// TIA Portal project "RUNNING_ A_PUMP" (V16)

(* hardware
DEVICE "S7-1200 station_1"  S7-1200 Station
   slot 0: "Rack_0"  S7-1200 Rack  Rack  V1.0
   slot 1: "PLC_1"  CPU 1214C DC/DC/DC  6ES7 214-1AG40-0XB0  V4.4
   slot 2: "AI 4x13BIT/AQ 2x14BIT_1"  6ES7 234-4HE32-0XB0  V2.1
*)

// ===== PLC "PLC_1"  CPU 1214C DC/DC/DC =====

VAR_GLOBAL   // PLC tag table "INPUTS&OUTPUT'"
   "START" AT %I0.1 : Bool;
   "PUMP" AT %Q0.0 : Bool;
   "PRESSURE_SENSOR" AT %IW64 : Int;
   "STORE_MEM" AT %MD30 : DInt;
   "MEM" AT %MD20 : DWord;
   "FLOW_VALVE_MEM" AT %MD24 : DWord;
   "FLOW_VALVE" AT %QW96 : Int;
END_VAR

ORGANIZATION_BLOCK "Main"   // OB1, LAD, ProgramCycle
TITLE = "Main Program Sweep (Cycle)"
{ S7_Optimized_Access := 'TRUE' }
VERSION : 0.1
   VAR_INPUT
      Initial_Call : Bool;   // Initial call of this OB
      Remanence : Bool;   // =True, if remanent data are available
   END_VAR
BEGIN

REGION Network 1
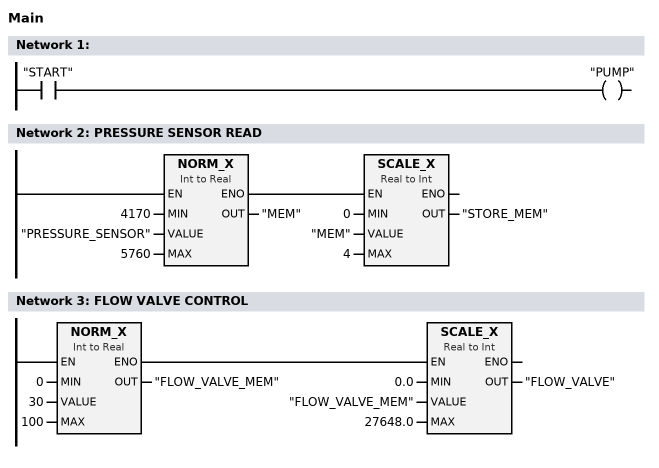
   RUNG wire#powerrail
      Contact( "START" )
      Coil( "PUMP" )
   END_RUNG
   // the same network as SCL:
   "PUMP" := "START";
END_REGION

REGION Network 2: PRESSURE SENSOR READ
   RUNG wire#powerrail
      { S7_Templates := "[SrcType := Int, DestType := Real]" } Normalize(min := 4170, value := "PRESSURE_SENSOR", max := 5760, out => "MEM")
      { S7_Templates := "[SrcType := Real, DestType := Int]" } Scale(min := 0, value := "MEM", max := 4, out => "STORE_MEM")
   END_RUNG
   // the same network as SCL:
   "MEM" := NORM_X(MIN := 4170, VALUE := "PRESSURE_SENSOR", MAX := 5760);
   "STORE_MEM" := SCALE_X(MIN := 0, VALUE := "MEM", MAX := 4);
END_REGION

REGION Network 3: FLOW VALVE CONTROL
   RUNG wire#powerrail
      { S7_Templates := "[SrcType := Int, DestType := Real]" } Normalize(min := 0, value := 30, max := 100, out => "FLOW_VALVE_MEM")
      { S7_Templates := "[SrcType := Real, DestType := Int]" } Scale(min := 0.0, value := "FLOW_VALVE_MEM", max := 27648.0, out => "FLOW_VALVE")
   END_RUNG
   // the same network as SCL:
   "FLOW_VALVE_MEM" := NORM_X(MIN := 0, VALUE := 30, MAX := 100);
   "FLOW_VALVE" := SCALE_X(MIN := 0.0, VALUE := "FLOW_VALVE_MEM", MAX := 27648.0);
END_REGION
END_ORGANIZATION_BLOCK